{attribute 'qualified_only'}
VAR_GLOBAL
	fDrumD : REAL := 0.475; //m
	fGearRatio : REAL := 1/20;
	//fMdisplacement	: REAL := 
	
END_VAR

(* stored: Version 1.1.0.1, ProductVersion 3.1.4024.12
   GVL CONSTANTS: Id {6656d0c1-0201-436e-b64b-6c1a30486286} *)
